FUNCTION_BLOCK FB_ClearPrechargeFailure
VAR_INPUT
END_VAR
VAR_OUTPUT
END_VAR
VAR
		send_message : PTC_Send_Message;
		fbTimer : TON;
END_VAR

send_message(ID := E_PTC_TX_ID.MAIN_FSM, Command := E_PTC_TX_Command.Clear_PreCharge_Failure, CAN_OUTPUTS := GVL_PT.CAN_OUTPUTS, CAN_INPUTS := GVL_PT.CAN_INPUTS);

END_FUNCTION_BLOCK

(* stored: Version 1.1.0.1
   POU FB_ClearPrechargeFailure: Id {aadba7ec-39bc-458a-8ca6-7ffc5beb20b0}, SpecialFunc None *)
